PROGRAM MAIN
VAR
	bTest				: BOOL;
	sTest				: STRING;
	
	bInput1				: BOOL;
	bOutput1			: BOOL;
END_VAR

IF bTest THEN
	sTest := 'Pull Test';
END_IF

Prg_Git();

END_PROGRAM

(* stored: Version 1.1.0.1, ProductVersion 3.1.4024.12
   POU MAIN: Id {8527cb53-8841-422c-b247-0d3122bcffe8}, SpecialFunc None *)
